TYPE U_XTS_STATION_STATE :
UNION
  stState             : ARRAY[1..MAX_STATION] OF ST_STATION_STATE;

  byState   AT %I*    : ARRAY[1..MAX_STATION] OF
                        ARRAY[1..SIZEOF(ST_STATION_STATE)] OF BYTE;
END_UNION
END_TYPE

(* stored: Version 1.1.0.1
   DUT U_XTS_STATION_STATE: Id {8d0bcd4b-dc0e-4310-825c-d0f4f8f94f49} *)
